{attribute 'GeneratedUsingTerminal: KL9900-0062'}
{attribute addProperty BoxType "KL9900-0062"}
{attribute addProperty Id "Channel_1AT %I*Channel_65B766000"}
{attribute addProperty CRC "3864242369"}
{attribute addProperty Size "0"}
TYPE KL_E653A8C1 :
STRUCT
	{attribute addProperty Name "Channel_1"}
	Channel_1 : Channel_65B76600;
END_STRUCT
END_TYPE

(* stored: Version 1.2.0.0, ProductVersion 3.1.4024.9
   DUT KL_E653A8C1: Id {1234e83a-d105-4862-9665-67cff71d5827} *)
